PROGRAM PRG_Diagnostic
VAR
	i: UDINT;
	StAlr	 : ARRAY[0..CNC.NUM_STATIONS+4] OF ARRAY[0..CNC.NUM_MAX_STATION_ALARMS-1] OF BOOL;
	fbEVSt00 : ARRAY[0..CNC.NUM_MAX_MANUALS_00-1] OF FB_PneumaticActuator_2EV_Diagnostic;
	fbEVSt01 : ARRAY[0..CNC.NUM_MAX_MANUALS_01-1] OF FB_PneumaticActuator_2EV_Diagnostic;
	fbEVSt02 : ARRAY[0..CNC.NUM_MAX_MANUALS_02-1] OF FB_PneumaticActuator_2EV_Diagnostic;
	fbEVSt03 : ARRAY[0..CNC.NUM_MAX_MANUALS_03-1] OF FB_PneumaticActuator_2EV_Diagnostic;
	fbEVSt04 : ARRAY[0..CNC.NUM_MAX_MANUALS_04-1] OF FB_PneumaticActuator_2EV_Diagnostic;
	fbEVSt05 : ARRAY[0..CNC.NUM_MAX_MANUALS_05-1] OF FB_PneumaticActuator_2EV_Diagnostic;
	fbEVSt06 : ARRAY[0..CNC.NUM_MAX_MANUALS_06-1] OF FB_PneumaticActuator_2EV_Diagnostic;
	fbEVSt07 : ARRAY[0..CNC.NUM_MAX_MANUALS_07-1] OF FB_PneumaticActuator_2EV_Diagnostic;
	fbEVSt08 : ARRAY[0..CNC.NUM_MAX_MANUALS_08-1] OF FB_PneumaticActuator_2EV_Diagnostic;
	fbEVSt09 : ARRAY[0..CNC.NUM_MAX_MANUALS_09-1] OF FB_PneumaticActuator_2EV_Diagnostic;
	fbEVSt10 : ARRAY[0..CNC.NUM_MAX_MANUALS_10-1] OF FB_PneumaticActuator_2EV_Diagnostic;
	fbEVSt11 : ARRAY[0..CNC.NUM_MAX_MANUALS_11-1] OF FB_PneumaticActuator_2EV_Diagnostic;
	fbEVSt12 : ARRAY[0..CNC.NUM_MAX_MANUALS_12-1] OF FB_PneumaticActuator_2EV_Diagnostic;
	fbEVSt13 : ARRAY[0..CNC.NUM_MAX_MANUALS_13-1] OF FB_PneumaticActuator_2EV_Diagnostic;	
END_VAR

A_01_EVDiagnostic();
A_02_EVDiagnostic();
A_03_EVDiagnostic();
A_04_EVDiagnostic();
A_05_EVDiagnostic();
A_06_EVDiagnostic();
A_07_EVDiagnostic();
A_08_EVDiagnostic();
A_09_EVDiagnostic();
A_10_EVDiagnostic();
A_11_EVDiagnostic();
A_12_EVDiagnostic();
A_13_EVDiagnostic();

A_01_Alarms();

ACTION A_00_Alarms:
FOR i:= 0 TO CNC.NUM_MAX_STATION_ALARMS -1 DO 
	StAlr[0][i] := PRG_EventManagement._PMCEventCollectors._CheckFanucPMCActiveAlarmList_St00_Alr._PMCEvents[i].bRaised;
END_FOR

HMI.St0.EVInfo[64].Error := PRG_Diagnostic.fbEVSt00[0].Q_eStatus = eEV_Status.MovingForward AND StAlr[1][0];		
HMI.St0.EVInfo[65].Error := PRG_Diagnostic.fbEVSt00[0].Q_eStatus = eEV_Status.MovingBackward AND StAlr[1][0];
HMI.St0.EVInfo[64].Error := PRG_Diagnostic.fbEVSt00[1].Q_eStatus = eEV_Status.MovingForward AND StAlr[1][0];
HMI.St0.EVInfo[65].Error := PRG_Diagnostic.fbEVSt00[1].Q_eStatus = eEV_Status.MovingBackward AND StAlr[1][0]; 
      
HMI.St0.EVInfo[66].dTime := PRG_Diagnostic.fbEVSt00[0].Q_tElapsedTimeFwd;		
HMI.St0.EVInfo[67].dTime := PRG_Diagnostic.fbEVSt00[0].Q_tElapsedTimeBwd;
HMI.St0.EVInfo[66].dTime := PRG_Diagnostic.fbEVSt00[1].Q_tElapsedTimeFwd;
HMI.St0.EVInfo[67].dTime := PRG_Diagnostic.fbEVSt00[1].Q_tElapsedTimeBwd;
END_ACTION

ACTION A_00_EVDiagnostic:
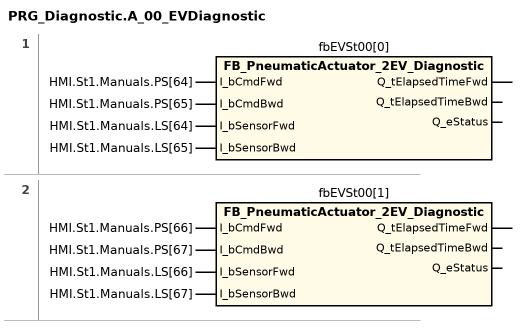
// NETWORK 1
fbEVSt00[0](
    I_bCmdFwd := HMI.St1.Manuals.PS[64],
    I_bCmdBwd := HMI.St1.Manuals.PS[65],
    I_bSensorFwd := HMI.St1.Manuals.LS[64],
    I_bSensorBwd := HMI.St1.Manuals.LS[65]); // FB_PneumaticActuator_2EV_Diagnostic

// NETWORK 2
fbEVSt00[1](
    I_bCmdFwd := HMI.St1.Manuals.PS[66],
    I_bCmdBwd := HMI.St1.Manuals.PS[67],
    I_bSensorFwd := HMI.St1.Manuals.LS[66],
    I_bSensorBwd := HMI.St1.Manuals.LS[67]); // FB_PneumaticActuator_2EV_Diagnostic
END_ACTION

ACTION A_01_Alarms:
FOR i:= 0 TO CNC.NUM_MAX_STATION_ALARMS -1 DO 
	StAlr[1][i] := PRG_EventManagement._PMCEventCollectors._CheckFanucPMCActiveAlarmList_St01_Alr._PMCEvents[i].bRaised;
END_FOR

HMI.St1.EVInfo[32].Error := PRG_Diagnostic.fbEVSt01[0].Q_eStatus = eEV_Status.MovingForward AND StAlr[1][0];		
HMI.St1.EVInfo[33].Error := PRG_Diagnostic.fbEVSt01[0].Q_eStatus = eEV_Status.MovingBackward AND StAlr[1][0];
HMI.St1.EVInfo[34].Error := PRG_Diagnostic.fbEVSt01[1].Q_eStatus = eEV_Status.MovingForward AND StAlr[1][0];
HMI.St1.EVInfo[35].Error := PRG_Diagnostic.fbEVSt01[1].Q_eStatus = eEV_Status.MovingBackward AND StAlr[1][0]; 
HMI.St1.EVInfo[36].Error := PRG_Diagnostic.fbEVSt01[2].Q_eStatus = eEV_Status.MovingForward AND StAlr[1][0];		
HMI.St1.EVInfo[37].Error := PRG_Diagnostic.fbEVSt01[2].Q_eStatus = eEV_Status.MovingBackward AND StAlr[1][0]; 
HMI.St1.EVInfo[25].Error := PRG_Diagnostic.fbEVSt01[3].Q_eStatus = eEV_Status.MovingForward AND StAlr[1][0];		
HMI.St1.EVInfo[26].Error := PRG_Diagnostic.fbEVSt01[3].Q_eStatus = eEV_Status.MovingBackward AND StAlr[1][0]; 

HMI.St1.EVInfo[32].dTime := PRG_Diagnostic.fbEVSt01[0].Q_tElapsedTimeFwd;		
HMI.St1.EVInfo[33].dTime := PRG_Diagnostic.fbEVSt01[0].Q_tElapsedTimeBwd;
HMI.St1.EVInfo[34].dTime := PRG_Diagnostic.fbEVSt01[1].Q_tElapsedTimeFwd;
HMI.St1.EVInfo[35].dTime := PRG_Diagnostic.fbEVSt01[1].Q_tElapsedTimeBwd;
HMI.St1.EVInfo[36].dTime := PRG_Diagnostic.fbEVSt01[2].Q_tElapsedTimeFwd;		
HMI.St1.EVInfo[37].dTime := PRG_Diagnostic.fbEVSt01[2].Q_tElapsedTimeBwd;
HMI.St1.EVInfo[25].dTime := PRG_Diagnostic.fbEVSt01[3].Q_tElapsedTimeFwd;		
HMI.St1.EVInfo[26].dTime := PRG_Diagnostic.fbEVSt01[3].Q_tElapsedTimeBwd;
END_ACTION

ACTION A_01_EVDiagnostic:
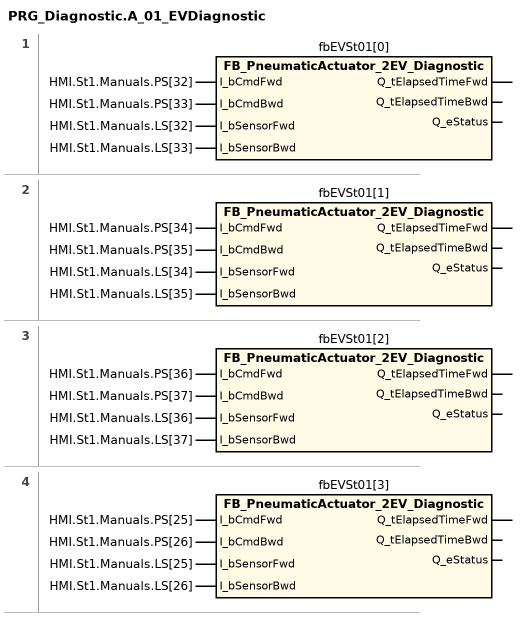
// NETWORK 1
fbEVSt01[0](
    I_bCmdFwd := HMI.St1.Manuals.PS[32],
    I_bCmdBwd := HMI.St1.Manuals.PS[33],
    I_bSensorFwd := HMI.St1.Manuals.LS[32],
    I_bSensorBwd := HMI.St1.Manuals.LS[33]); // FB_PneumaticActuator_2EV_Diagnostic

// NETWORK 2
fbEVSt01[1](
    I_bCmdFwd := HMI.St1.Manuals.PS[34],
    I_bCmdBwd := HMI.St1.Manuals.PS[35],
    I_bSensorFwd := HMI.St1.Manuals.LS[34],
    I_bSensorBwd := HMI.St1.Manuals.LS[35]); // FB_PneumaticActuator_2EV_Diagnostic

// NETWORK 3
fbEVSt01[2](
    I_bCmdFwd := HMI.St1.Manuals.PS[36],
    I_bCmdBwd := HMI.St1.Manuals.PS[37],
    I_bSensorFwd := HMI.St1.Manuals.LS[36],
    I_bSensorBwd := HMI.St1.Manuals.LS[37]); // FB_PneumaticActuator_2EV_Diagnostic

// NETWORK 4
fbEVSt01[3](
    I_bCmdFwd := HMI.St1.Manuals.PS[25],
    I_bCmdBwd := HMI.St1.Manuals.PS[26],
    I_bSensorFwd := HMI.St1.Manuals.LS[25],
    I_bSensorBwd := HMI.St1.Manuals.LS[26]); // FB_PneumaticActuator_2EV_Diagnostic
END_ACTION

ACTION A_02_Alarms:
FOR i:= 0 TO CNC.NUM_MAX_STATION_ALARMS -1 DO 
	StAlr[2][i] := PRG_EventManagement._PMCEventCollectors._CheckFanucPMCActiveAlarmList_St02_Alr._PMCEvents[i].bRaised;
END_FOR

HMI.St2.EVInfo[32].Error := PRG_Diagnostic.fbEVSt02[0].Q_eStatus = eEV_Status.MovingForward  AND StAlr[2][0];		
HMI.St2.EVInfo[33].Error := PRG_Diagnostic.fbEVSt02[0].Q_eStatus = eEV_Status.MovingBackward AND StAlr[2][0];
HMI.St2.EVInfo[34].Error := PRG_Diagnostic.fbEVSt02[1].Q_eStatus = eEV_Status.MovingForward  AND StAlr[2][0];
HMI.St2.EVInfo[35].Error := PRG_Diagnostic.fbEVSt02[1].Q_eStatus = eEV_Status.MovingBackward AND StAlr[2][0]; 
                                                  
HMI.St2.EVInfo[32].dTime := PRG_Diagnostic.fbEVSt02[0].Q_tElapsedTimeFwd;		
HMI.St2.EVInfo[33].dTime := PRG_Diagnostic.fbEVSt02[0].Q_tElapsedTimeBwd;
HMI.St2.EVInfo[34].dTime := PRG_Diagnostic.fbEVSt02[1].Q_tElapsedTimeFwd;
HMI.St2.EVInfo[35].dTime := PRG_Diagnostic.fbEVSt02[1].Q_tElapsedTimeBwd;
END_ACTION

ACTION A_02_EVDiagnostic:
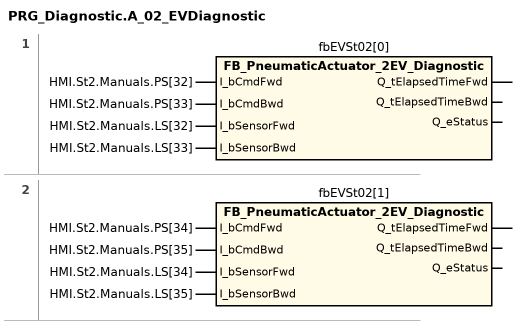
// NETWORK 1
fbEVSt02[0](
    I_bCmdFwd := HMI.St2.Manuals.PS[32],
    I_bCmdBwd := HMI.St2.Manuals.PS[33],
    I_bSensorFwd := HMI.St2.Manuals.LS[32],
    I_bSensorBwd := HMI.St2.Manuals.LS[33]); // FB_PneumaticActuator_2EV_Diagnostic

// NETWORK 2
fbEVSt02[1](
    I_bCmdFwd := HMI.St2.Manuals.PS[34],
    I_bCmdBwd := HMI.St2.Manuals.PS[35],
    I_bSensorFwd := HMI.St2.Manuals.LS[34],
    I_bSensorBwd := HMI.St2.Manuals.LS[35]); // FB_PneumaticActuator_2EV_Diagnostic
END_ACTION

ACTION A_03_Alarms:
FOR i:= 0 TO CNC.NUM_MAX_STATION_ALARMS -1 DO 
	StAlr[3][i] := PRG_EventManagement._PMCEventCollectors._CheckFanucPMCActiveAlarmList_St03_Alr._PMCEvents[i].bRaised;
END_FOR

HMI.St3.EVInfo[33].Error := PRG_Diagnostic.fbEVSt03[0].Q_eStatus = eEV_Status.MovingForward  AND StAlr[3][0];		
HMI.St3.EVInfo[32].Error := PRG_Diagnostic.fbEVSt03[0].Q_eStatus = eEV_Status.MovingBackward AND StAlr[3][0];
      
HMI.St3.EVInfo[33].dTime := PRG_Diagnostic.fbEVSt03[0].Q_tElapsedTimeFwd;		
HMI.St3.EVInfo[32].dTime := PRG_Diagnostic.fbEVSt03[0].Q_tElapsedTimeBwd;
END_ACTION

ACTION A_03_EVDiagnostic:
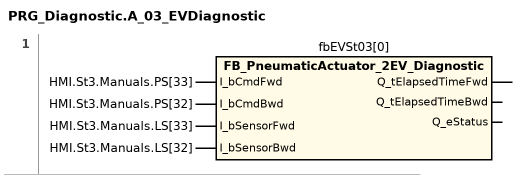
// NETWORK 1
fbEVSt03[0](
    I_bCmdFwd := HMI.St3.Manuals.PS[33],
    I_bCmdBwd := HMI.St3.Manuals.PS[32],
    I_bSensorFwd := HMI.St3.Manuals.LS[33],
    I_bSensorBwd := HMI.St3.Manuals.LS[32]); // FB_PneumaticActuator_2EV_Diagnostic
END_ACTION

ACTION A_04_Alarms:
FOR i:= 0 TO CNC.NUM_MAX_STATION_ALARMS -1 DO 
	StAlr[4][i] := PRG_EventManagement._PMCEventCollectors._CheckFanucPMCActiveAlarmList_St04_Alr._PMCEvents[i].bRaised;
END_FOR

HMI.St4.EVInfo[36].Error := PRG_Diagnostic.fbEVSt04[2].Q_eStatus = eEV_Status.MovingForward  AND StAlr[4][0];
HMI.St4.EVInfo[37].Error := PRG_Diagnostic.fbEVSt04[2].Q_eStatus = eEV_Status.MovingBackward AND StAlr[4][0]; 
HMI.St4.EVInfo[38].Error := PRG_Diagnostic.fbEVSt04[3].Q_eStatus = eEV_Status.MovingForward  AND StAlr[4][0];		
HMI.St4.EVInfo[39].Error := PRG_Diagnostic.fbEVSt04[3].Q_eStatus = eEV_Status.MovingBackward AND StAlr[4][0]; 
                                                  
HMI.St4.EVInfo[36].dTime := PRG_Diagnostic.fbEVSt04[2].Q_tElapsedTimeFwd;		
HMI.St4.EVInfo[37].dTime := PRG_Diagnostic.fbEVSt04[2].Q_tElapsedTimeBwd;
HMI.St4.EVInfo[38].dTime := PRG_Diagnostic.fbEVSt04[3].Q_tElapsedTimeFwd;
HMI.St4.EVInfo[39].dTime := PRG_Diagnostic.fbEVSt04[3].Q_tElapsedTimeBwd;
END_ACTION

ACTION A_04_EVDiagnostic:
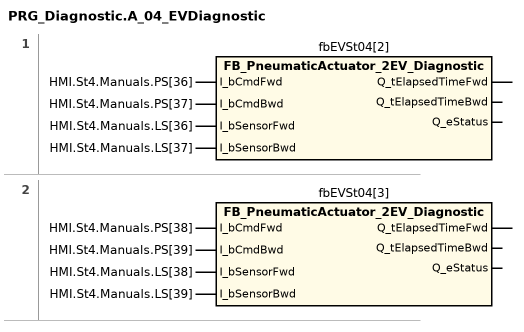
// NETWORK 1
fbEVSt04[2](
    I_bCmdFwd := HMI.St4.Manuals.PS[36],
    I_bCmdBwd := HMI.St4.Manuals.PS[37],
    I_bSensorFwd := HMI.St4.Manuals.LS[36],
    I_bSensorBwd := HMI.St4.Manuals.LS[37]); // FB_PneumaticActuator_2EV_Diagnostic

// NETWORK 2
fbEVSt04[3](
    I_bCmdFwd := HMI.St4.Manuals.PS[38],
    I_bCmdBwd := HMI.St4.Manuals.PS[39],
    I_bSensorFwd := HMI.St4.Manuals.LS[38],
    I_bSensorBwd := HMI.St4.Manuals.LS[39]); // FB_PneumaticActuator_2EV_Diagnostic
END_ACTION

ACTION A_05_Alarms:
FOR i:= 0 TO CNC.NUM_MAX_STATION_ALARMS -1 DO 
	StAlr[5][i] := PRG_EventManagement._PMCEventCollectors._CheckFanucPMCActiveAlarmList_St05_Alr._PMCEvents[i].bRaised;
END_FOR

HMI.St5.EVInfo[40].Error := PRG_Diagnostic.fbEVSt05[4].Q_eStatus  = eEV_Status.MovingForward  AND StAlr[5][0];		
HMI.St5.EVInfo[41].Error := PRG_Diagnostic.fbEVSt05[4].Q_eStatus  = eEV_Status.MovingBackward AND StAlr[5][0];
HMI.St5.EVInfo[64].Error := PRG_Diagnostic.fbEVSt05[16].Q_eStatus = eEV_Status.MovingForward  AND StAlr[5][0];
HMI.St5.EVInfo[65].Error := PRG_Diagnostic.fbEVSt05[16].Q_eStatus = eEV_Status.MovingBackward AND StAlr[5][0]; 
HMI.St5.EVInfo[66].Error := PRG_Diagnostic.fbEVSt05[17].Q_eStatus = eEV_Status.MovingForward  AND StAlr[5][0];		
HMI.St5.EVInfo[67].Error := PRG_Diagnostic.fbEVSt05[17].Q_eStatus = eEV_Status.MovingBackward AND StAlr[5][0]; 
                                                  
HMI.St5.EVInfo[40].dTime := PRG_Diagnostic.fbEVSt05[4].Q_tElapsedTimeFwd;		
HMI.St5.EVInfo[41].dTime := PRG_Diagnostic.fbEVSt05[4].Q_tElapsedTimeBwd;
HMI.St5.EVInfo[64].dTime := PRG_Diagnostic.fbEVSt05[16].Q_tElapsedTimeFwd;
HMI.St5.EVInfo[65].dTime := PRG_Diagnostic.fbEVSt05[16].Q_tElapsedTimeBwd;
HMI.St5.EVInfo[66].dTime := PRG_Diagnostic.fbEVSt05[17].Q_tElapsedTimeFwd;		
HMI.St5.EVInfo[67].dTime := PRG_Diagnostic.fbEVSt05[17].Q_tElapsedTimeBwd;
END_ACTION

ACTION A_05_EVDiagnostic:
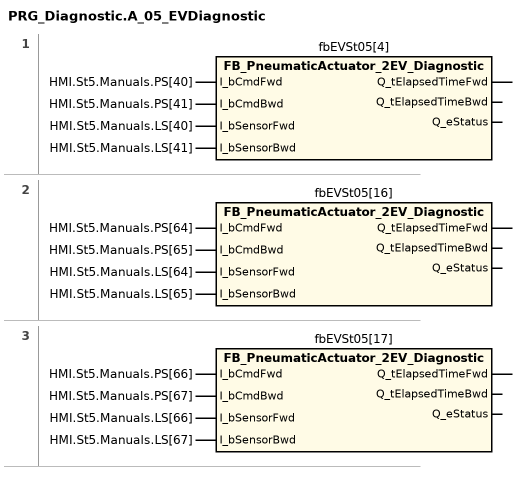
// NETWORK 1
fbEVSt05[4](
    I_bCmdFwd := HMI.St5.Manuals.PS[40],
    I_bCmdBwd := HMI.St5.Manuals.PS[41],
    I_bSensorFwd := HMI.St5.Manuals.LS[40],
    I_bSensorBwd := HMI.St5.Manuals.LS[41]); // FB_PneumaticActuator_2EV_Diagnostic

// NETWORK 2
fbEVSt05[16](
    I_bCmdFwd := HMI.St5.Manuals.PS[64],
    I_bCmdBwd := HMI.St5.Manuals.PS[65],
    I_bSensorFwd := HMI.St5.Manuals.LS[64],
    I_bSensorBwd := HMI.St5.Manuals.LS[65]); // FB_PneumaticActuator_2EV_Diagnostic

// NETWORK 3
fbEVSt05[17](
    I_bCmdFwd := HMI.St5.Manuals.PS[66],
    I_bCmdBwd := HMI.St5.Manuals.PS[67],
    I_bSensorFwd := HMI.St5.Manuals.LS[66],
    I_bSensorBwd := HMI.St5.Manuals.LS[67]); // FB_PneumaticActuator_2EV_Diagnostic
END_ACTION

ACTION A_06_Alarms:
FOR i:= 0 TO CNC.NUM_MAX_STATION_ALARMS -1 DO 
	StAlr[6][i] := PRG_EventManagement._PMCEventCollectors._CheckFanucPMCActiveAlarmList_St06_Alr._PMCEvents[i].bRaised;
END_FOR

HMI.St6.EVInfo[40].Error := PRG_Diagnostic.fbEVSt06[4].Q_eStatus = eEV_Status.MovingForward  AND StAlr[6][0];		
HMI.St6.EVInfo[41].Error := PRG_Diagnostic.fbEVSt06[4].Q_eStatus = eEV_Status.MovingBackward AND StAlr[6][0]; 

HMI.St6.EVInfo[40].dTime := PRG_Diagnostic.fbEVSt06[4].Q_tElapsedTimeFwd;		
HMI.St6.EVInfo[41].dTime := PRG_Diagnostic.fbEVSt06[4].Q_tElapsedTimeBwd;
END_ACTION

ACTION A_06_EVDiagnostic:
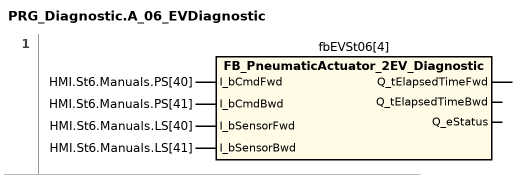
// NETWORK 1
fbEVSt06[4](
    I_bCmdFwd := HMI.St6.Manuals.PS[40],
    I_bCmdBwd := HMI.St6.Manuals.PS[41],
    I_bSensorFwd := HMI.St6.Manuals.LS[40],
    I_bSensorBwd := HMI.St6.Manuals.LS[41]); // FB_PneumaticActuator_2EV_Diagnostic
END_ACTION

ACTION A_07_Alarms:
FOR i:= 0 TO CNC.NUM_MAX_STATION_ALARMS -1 DO 
	StAlr[7][i] := PRG_EventManagement._PMCEventCollectors._CheckFanucPMCActiveAlarmList_St07_Alr._PMCEvents[i].bRaised;
END_FOR

HMI.St1.EVInfo[40].Error := PRG_Diagnostic.fbEVSt07[4].Q_eStatus = eEV_Status.MovingForward  AND StAlr[7][0];		
HMI.St1.EVInfo[41].Error := PRG_Diagnostic.fbEVSt07[4].Q_eStatus = eEV_Status.MovingBackward AND StAlr[7][0];

HMI.St1.EVInfo[40].dTime := PRG_Diagnostic.fbEVSt07[4].Q_tElapsedTimeFwd;		
HMI.St1.EVInfo[41].dTime := PRG_Diagnostic.fbEVSt07[4].Q_tElapsedTimeBwd;
END_ACTION

ACTION A_07_EVDiagnostic:
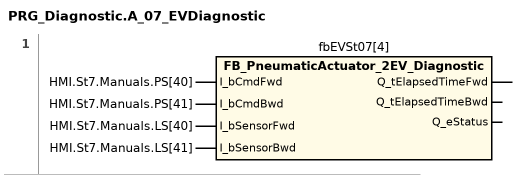
// NETWORK 1
fbEVSt07[4](
    I_bCmdFwd := HMI.St7.Manuals.PS[40],
    I_bCmdBwd := HMI.St7.Manuals.PS[41],
    I_bSensorFwd := HMI.St7.Manuals.LS[40],
    I_bSensorBwd := HMI.St7.Manuals.LS[41]); // FB_PneumaticActuator_2EV_Diagnostic
END_ACTION

ACTION A_08_Alarms:
FOR i:= 0 TO CNC.NUM_MAX_STATION_ALARMS -1 DO 
	StAlr[8][i] := PRG_EventManagement._PMCEventCollectors._CheckFanucPMCActiveAlarmList_St08_Alr._PMCEvents[i].bRaised;
END_FOR

HMI.St8.EVInfo[40].Error := PRG_Diagnostic.fbEVSt08[0].Q_eStatus = eEV_Status.MovingForward  AND StAlr[8][0];		
HMI.St8.EVInfo[41].Error := PRG_Diagnostic.fbEVSt08[0].Q_eStatus = eEV_Status.MovingBackward AND StAlr[8][0];

HMI.St8.EVInfo[40].dTime := PRG_Diagnostic.fbEVSt08[0].Q_tElapsedTimeFwd;		
HMI.St8.EVInfo[41].dTime := PRG_Diagnostic.fbEVSt08[0].Q_tElapsedTimeBwd;
END_ACTION

ACTION A_08_EVDiagnostic:
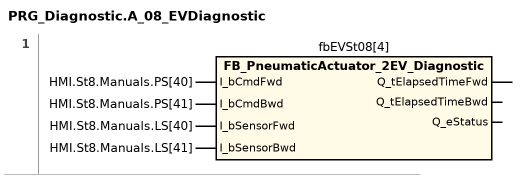
// NETWORK 1
fbEVSt08[4](
    I_bCmdFwd := HMI.St8.Manuals.PS[40],
    I_bCmdBwd := HMI.St8.Manuals.PS[41],
    I_bSensorFwd := HMI.St8.Manuals.LS[40],
    I_bSensorBwd := HMI.St8.Manuals.LS[41]); // FB_PneumaticActuator_2EV_Diagnostic
END_ACTION

ACTION A_09_Alarms:
FOR i:= 0 TO CNC.NUM_MAX_STATION_ALARMS -1 DO 
	StAlr[9][i] := PRG_EventManagement._PMCEventCollectors._CheckFanucPMCActiveAlarmList_St09_Alr._PMCEvents[i].bRaised;
END_FOR

HMI.St9.EVInfo[40].Error := PRG_Diagnostic.fbEVSt09[4].Q_eStatus = eEV_Status.MovingForward  AND StAlr[1][0];		
HMI.St9.EVInfo[41].Error := PRG_Diagnostic.fbEVSt09[4].Q_eStatus = eEV_Status.MovingBackward AND StAlr[1][0];

HMI.St9.EVInfo[40].dTime := PRG_Diagnostic.fbEVSt09[4].Q_tElapsedTimeFwd;		
HMI.St9.EVInfo[41].dTime := PRG_Diagnostic.fbEVSt09[4].Q_tElapsedTimeBwd;
END_ACTION

ACTION A_09_EVDiagnostic:
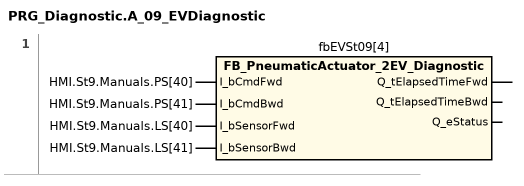
// NETWORK 1
fbEVSt09[4](
    I_bCmdFwd := HMI.St9.Manuals.PS[40],
    I_bCmdBwd := HMI.St9.Manuals.PS[41],
    I_bSensorFwd := HMI.St9.Manuals.LS[40],
    I_bSensorBwd := HMI.St9.Manuals.LS[41]); // FB_PneumaticActuator_2EV_Diagnostic
END_ACTION

ACTION A_10_Alarms:
FOR i:= 0 TO CNC.NUM_MAX_STATION_ALARMS -1 DO 
	StAlr[10][i] := PRG_EventManagement._PMCEventCollectors._CheckFanucPMCActiveAlarmList_St10_Alr._PMCEvents[i].bRaised;
END_FOR

HMI.St10.EVInfo[40].Error := PRG_Diagnostic.fbEVSt10[4].Q_eStatus = eEV_Status.MovingForward   AND StAlr[10][0];		
HMI.St10.EVInfo[41].Error := PRG_Diagnostic.fbEVSt10[4].Q_eStatus = eEV_Status.MovingBackward  AND StAlr[10][0];
HMI.St10.EVInfo[40].Error := PRG_Diagnostic.fbEVSt10[11].Q_eStatus = eEV_Status.MovingForward  AND StAlr[10][0];
HMI.St10.EVInfo[41].Error := PRG_Diagnostic.fbEVSt10[11].Q_eStatus = eEV_Status.MovingBackward AND StAlr[10][0]; 
                                                  
HMI.St10.EVInfo[54].dTime := PRG_Diagnostic.fbEVSt10[4].Q_tElapsedTimeFwd;		
HMI.St10.EVInfo[55].dTime := PRG_Diagnostic.fbEVSt10[4].Q_tElapsedTimeBwd;
HMI.St10.EVInfo[54].dTime := PRG_Diagnostic.fbEVSt10[11].Q_tElapsedTimeFwd;
HMI.St10.EVInfo[55].dTime := PRG_Diagnostic.fbEVSt10[11].Q_tElapsedTimeBwd;
END_ACTION

ACTION A_10_EVDiagnostic:
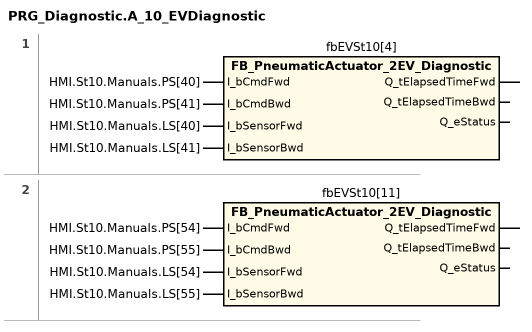
// NETWORK 1
fbEVSt10[4](
    I_bCmdFwd := HMI.St10.Manuals.PS[40],
    I_bCmdBwd := HMI.St10.Manuals.PS[41],
    I_bSensorFwd := HMI.St10.Manuals.LS[40],
    I_bSensorBwd := HMI.St10.Manuals.LS[41]); // FB_PneumaticActuator_2EV_Diagnostic

// NETWORK 2
fbEVSt10[11](
    I_bCmdFwd := HMI.St10.Manuals.PS[54],
    I_bCmdBwd := HMI.St10.Manuals.PS[55],
    I_bSensorFwd := HMI.St10.Manuals.LS[54],
    I_bSensorBwd := HMI.St10.Manuals.LS[55]); // FB_PneumaticActuator_2EV_Diagnostic
END_ACTION

ACTION A_11_Alarms:
FOR i:= 0 TO CNC.NUM_MAX_STATION_ALARMS -1 DO 
	StAlr[11][i] := PRG_EventManagement._PMCEventCollectors._CheckFanucPMCActiveAlarmList_St11_Alr._PMCEvents[i].bRaised;
END_FOR

HMI.St11.EVInfo[32].Error := PRG_Diagnostic.fbEVSt01[0].Q_eStatus = eEV_Status.MovingForward  AND StAlr[11][0];		
HMI.St11.EVInfo[33].Error := PRG_Diagnostic.fbEVSt01[0].Q_eStatus = eEV_Status.MovingBackward AND StAlr[11][0];
HMI.St11.EVInfo[34].Error := PRG_Diagnostic.fbEVSt01[1].Q_eStatus = eEV_Status.MovingForward  AND StAlr[11][0];
HMI.St11.EVInfo[35].Error := PRG_Diagnostic.fbEVSt01[1].Q_eStatus = eEV_Status.MovingBackward AND StAlr[11][0]; 

HMI.St11.EVInfo[32].dTime := PRG_Diagnostic.fbEVSt01[0].Q_tElapsedTimeFwd;		
HMI.St11.EVInfo[33].dTime := PRG_Diagnostic.fbEVSt01[0].Q_tElapsedTimeBwd;
HMI.St11.EVInfo[34].dTime := PRG_Diagnostic.fbEVSt01[1].Q_tElapsedTimeFwd;
HMI.St11.EVInfo[35].dTime := PRG_Diagnostic.fbEVSt01[1].Q_tElapsedTimeBwd;
END_ACTION

ACTION A_11_EVDiagnostic:
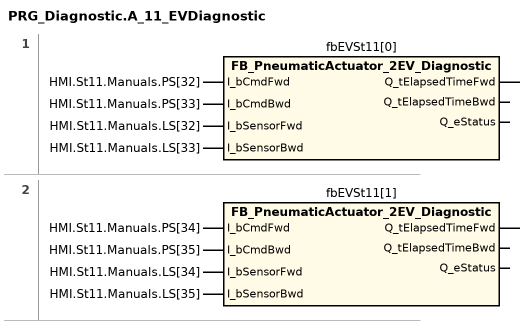
// NETWORK 1
fbEVSt11[0](
    I_bCmdFwd := HMI.St11.Manuals.PS[32],
    I_bCmdBwd := HMI.St11.Manuals.PS[33],
    I_bSensorFwd := HMI.St11.Manuals.LS[32],
    I_bSensorBwd := HMI.St11.Manuals.LS[33]); // FB_PneumaticActuator_2EV_Diagnostic

// NETWORK 2
fbEVSt11[1](
    I_bCmdFwd := HMI.St11.Manuals.PS[34],
    I_bCmdBwd := HMI.St11.Manuals.PS[35],
    I_bSensorFwd := HMI.St11.Manuals.LS[34],
    I_bSensorBwd := HMI.St11.Manuals.LS[35]); // FB_PneumaticActuator_2EV_Diagnostic
END_ACTION

ACTION A_12_Alarms:
FOR i:= 0 TO CNC.NUM_MAX_STATION_ALARMS -1 DO 
	StAlr[12][i] := PRG_EventManagement._PMCEventCollectors._CheckFanucPMCActiveAlarmList_St12_Alr._PMCEvents[i].bRaised;
END_FOR

HMI.St12.EVInfo[32].Error := PRG_Diagnostic.fbEVSt12[0].Q_eStatus = eEV_Status.MovingForward  AND StAlr[12][0];		
HMI.St12.EVInfo[33].Error := PRG_Diagnostic.fbEVSt12[0].Q_eStatus = eEV_Status.MovingBackward AND StAlr[12][0];
HMI.St12.EVInfo[34].Error := PRG_Diagnostic.fbEVSt12[1].Q_eStatus = eEV_Status.MovingForward  AND StAlr[12][0];
HMI.St12.EVInfo[35].Error := PRG_Diagnostic.fbEVSt12[1].Q_eStatus = eEV_Status.MovingBackward AND StAlr[12][0]; 
HMI.St12.EVInfo[36].Error := PRG_Diagnostic.fbEVSt12[2].Q_eStatus = eEV_Status.MovingForward  AND StAlr[12][0];		
HMI.St12.EVInfo[37].Error := PRG_Diagnostic.fbEVSt12[2].Q_eStatus = eEV_Status.MovingBackward AND StAlr[12][0];
HMI.St12.EVInfo[38].Error := PRG_Diagnostic.fbEVSt12[3].Q_eStatus = eEV_Status.MovingForward  AND StAlr[12][0];		
HMI.St12.EVInfo[39].Error := PRG_Diagnostic.fbEVSt12[3].Q_eStatus = eEV_Status.MovingBackward AND StAlr[12][0];
HMI.St12.EVInfo[40].Error := PRG_Diagnostic.fbEVSt12[4].Q_eStatus = eEV_Status.MovingForward  AND StAlr[12][0];		
HMI.St12.EVInfo[41].Error := PRG_Diagnostic.fbEVSt12[4].Q_eStatus = eEV_Status.MovingBackward AND StAlr[12][0]; 

HMI.St12.EVInfo[32].dTime := PRG_Diagnostic.fbEVSt12[0].Q_tElapsedTimeFwd;		
HMI.St12.EVInfo[33].dTime := PRG_Diagnostic.fbEVSt12[0].Q_tElapsedTimeBwd;
HMI.St12.EVInfo[34].dTime := PRG_Diagnostic.fbEVSt12[1].Q_tElapsedTimeFwd;
HMI.St12.EVInfo[35].dTime := PRG_Diagnostic.fbEVSt12[1].Q_tElapsedTimeBwd;
HMI.St12.EVInfo[36].dTime := PRG_Diagnostic.fbEVSt12[2].Q_tElapsedTimeFwd;		
HMI.St12.EVInfo[37].dTime := PRG_Diagnostic.fbEVSt12[2].Q_tElapsedTimeBwd;
HMI.St12.EVInfo[38].dTime := PRG_Diagnostic.fbEVSt12[3].Q_tElapsedTimeFwd;		
HMI.St12.EVInfo[39].dTime := PRG_Diagnostic.fbEVSt12[3].Q_tElapsedTimeBwd;
HMI.St12.EVInfo[40].dTime := PRG_Diagnostic.fbEVSt12[4].Q_tElapsedTimeFwd;		
HMI.St12.EVInfo[41].dTime := PRG_Diagnostic.fbEVSt12[4].Q_tElapsedTimeBwd;
END_ACTION

ACTION A_12_EVDiagnostic:
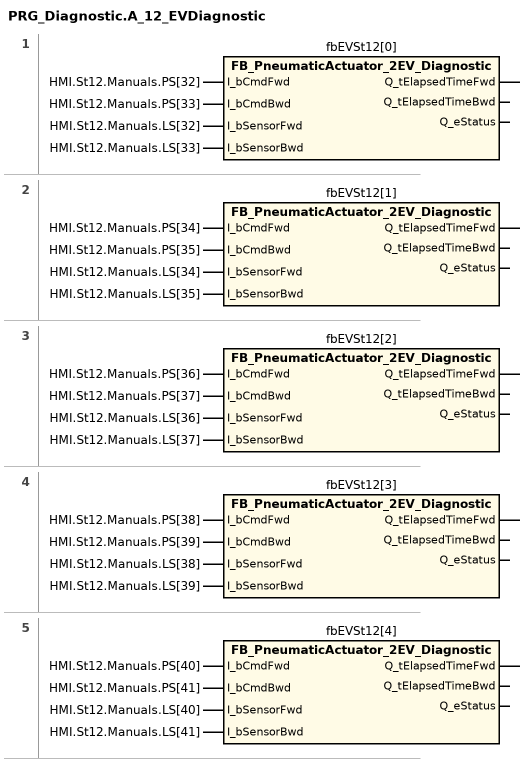
// NETWORK 1
fbEVSt12[0](
    I_bCmdFwd := HMI.St12.Manuals.PS[32],
    I_bCmdBwd := HMI.St12.Manuals.PS[33],
    I_bSensorFwd := HMI.St12.Manuals.LS[32],
    I_bSensorBwd := HMI.St12.Manuals.LS[33]); // FB_PneumaticActuator_2EV_Diagnostic

// NETWORK 2
fbEVSt12[1](
    I_bCmdFwd := HMI.St12.Manuals.PS[34],
    I_bCmdBwd := HMI.St12.Manuals.PS[35],
    I_bSensorFwd := HMI.St12.Manuals.LS[34],
    I_bSensorBwd := HMI.St12.Manuals.LS[35]); // FB_PneumaticActuator_2EV_Diagnostic

// NETWORK 3
fbEVSt12[2](
    I_bCmdFwd := HMI.St12.Manuals.PS[36],
    I_bCmdBwd := HMI.St12.Manuals.PS[37],
    I_bSensorFwd := HMI.St12.Manuals.LS[36],
    I_bSensorBwd := HMI.St12.Manuals.LS[37]); // FB_PneumaticActuator_2EV_Diagnostic

// NETWORK 4
fbEVSt12[3](
    I_bCmdFwd := HMI.St12.Manuals.PS[38],
    I_bCmdBwd := HMI.St12.Manuals.PS[39],
    I_bSensorFwd := HMI.St12.Manuals.LS[38],
    I_bSensorBwd := HMI.St12.Manuals.LS[39]); // FB_PneumaticActuator_2EV_Diagnostic

// NETWORK 5
fbEVSt12[4](
    I_bCmdFwd := HMI.St12.Manuals.PS[40],
    I_bCmdBwd := HMI.St12.Manuals.PS[41],
    I_bSensorFwd := HMI.St12.Manuals.LS[40],
    I_bSensorBwd := HMI.St12.Manuals.LS[41]); // FB_PneumaticActuator_2EV_Diagnostic
END_ACTION

ACTION A_13_Alarms:
FOR i:= 0 TO CNC.NUM_MAX_STATION_ALARMS -1 DO 
	StAlr[13][i] := PRG_EventManagement._PMCEventCollectors._CheckFanucPMCActiveAlarmList_St13_Alr._PMCEvents[i].bRaised;
END_FOR

HMI.St13.EVInfo[32].Error := PRG_Diagnostic.fbEVSt13[0].Q_eStatus = eEV_Status.MovingForward  AND StAlr[13][0];		
HMI.St13.EVInfo[33].Error := PRG_Diagnostic.fbEVSt13[0].Q_eStatus = eEV_Status.MovingBackward AND StAlr[13][0];
HMI.St13.EVInfo[34].Error := PRG_Diagnostic.fbEVSt13[1].Q_eStatus = eEV_Status.MovingForward  AND StAlr[13][0];
HMI.St13.EVInfo[35].Error := PRG_Diagnostic.fbEVSt13[1].Q_eStatus = eEV_Status.MovingBackward AND StAlr[13][0]; 
HMI.St13.EVInfo[36].Error := PRG_Diagnostic.fbEVSt13[2].Q_eStatus = eEV_Status.MovingForward  AND StAlr[13][0];		
HMI.St13.EVInfo[37].Error := PRG_Diagnostic.fbEVSt13[2].Q_eStatus = eEV_Status.MovingBackward AND StAlr[13][0]; 
HMI.St13.EVInfo[38].Error := PRG_Diagnostic.fbEVSt13[3].Q_eStatus = eEV_Status.MovingForward  AND StAlr[13][0];		
HMI.St13.EVInfo[39].Error := PRG_Diagnostic.fbEVSt13[3].Q_eStatus = eEV_Status.MovingBackward AND StAlr[13][0]; 

HMI.St13.EVInfo[32].dTime := PRG_Diagnostic.fbEVSt13[0].Q_tElapsedTimeFwd;		
HMI.St13.EVInfo[33].dTime := PRG_Diagnostic.fbEVSt13[0].Q_tElapsedTimeBwd;
HMI.St13.EVInfo[34].dTime := PRG_Diagnostic.fbEVSt13[1].Q_tElapsedTimeFwd;
HMI.St13.EVInfo[35].dTime := PRG_Diagnostic.fbEVSt13[1].Q_tElapsedTimeBwd;
HMI.St13.EVInfo[36].dTime := PRG_Diagnostic.fbEVSt13[2].Q_tElapsedTimeFwd;		
HMI.St13.EVInfo[37].dTime := PRG_Diagnostic.fbEVSt13[2].Q_tElapsedTimeBwd;
HMI.St13.EVInfo[38].dTime := PRG_Diagnostic.fbEVSt13[3].Q_tElapsedTimeFwd;		
HMI.St13.EVInfo[39].dTime := PRG_Diagnostic.fbEVSt13[3].Q_tElapsedTimeBwd;
END_ACTION

ACTION A_13_EVDiagnostic:
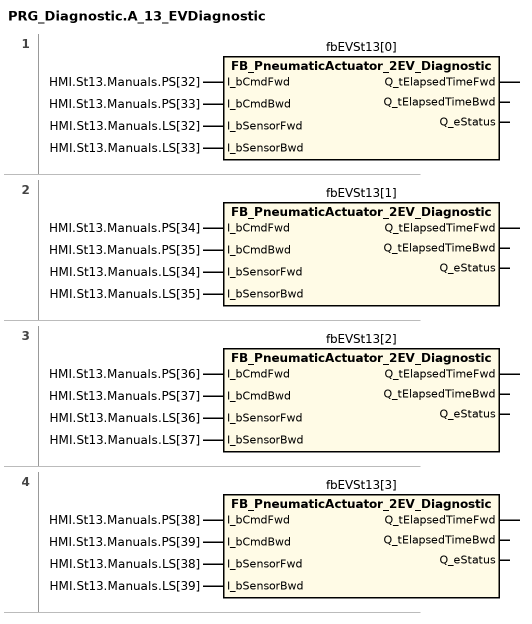
// NETWORK 1
fbEVSt13[0](
    I_bCmdFwd := HMI.St13.Manuals.PS[32],
    I_bCmdBwd := HMI.St13.Manuals.PS[33],
    I_bSensorFwd := HMI.St13.Manuals.LS[32],
    I_bSensorBwd := HMI.St13.Manuals.LS[33]); // FB_PneumaticActuator_2EV_Diagnostic

// NETWORK 2
fbEVSt13[1](
    I_bCmdFwd := HMI.St13.Manuals.PS[34],
    I_bCmdBwd := HMI.St13.Manuals.PS[35],
    I_bSensorFwd := HMI.St13.Manuals.LS[34],
    I_bSensorBwd := HMI.St13.Manuals.LS[35]); // FB_PneumaticActuator_2EV_Diagnostic

// NETWORK 3
fbEVSt13[2](
    I_bCmdFwd := HMI.St13.Manuals.PS[36],
    I_bCmdBwd := HMI.St13.Manuals.PS[37],
    I_bSensorFwd := HMI.St13.Manuals.LS[36],
    I_bSensorBwd := HMI.St13.Manuals.LS[37]); // FB_PneumaticActuator_2EV_Diagnostic

// NETWORK 4
fbEVSt13[3](
    I_bCmdFwd := HMI.St13.Manuals.PS[38],
    I_bCmdBwd := HMI.St13.Manuals.PS[39],
    I_bSensorFwd := HMI.St13.Manuals.LS[38],
    I_bSensorBwd := HMI.St13.Manuals.LS[39]); // FB_PneumaticActuator_2EV_Diagnostic
END_ACTION

END_PROGRAM

(* stored: Version 1.1.0.1, ProductVersion 3.1.4024.15
   POU PRG_Diagnostic: Id {adc91861-aa55-4305-bfac-bd2b856a148e}, SpecialFunc None
   Action A_00_Alarms: Id {18c0b9bd-8ae9-4423-847e-db8238966453}
   Action A_00_EVDiagnostic: Id {59c9defa-d32a-4095-aa94-e7b90637144f}
   Action A_01_Alarms: Id {24727d9b-13c9-4222-9961-ff712a4c9358}
   Action A_01_EVDiagnostic: Id {88fcfb40-2b85-4632-a930-2deb89fcff3e}
   Action A_02_Alarms: Id {b0148c85-5ccf-4e62-bb15-5fd4490b1a3a}
   Action A_02_EVDiagnostic: Id {488b1e0b-e364-4a56-868e-4b715e806523}
   Action A_03_Alarms: Id {dc5e5318-976e-4aff-905f-e35ce54c1fa3}
   Action A_03_EVDiagnostic: Id {c65fc63d-e765-4de2-a2b2-de392bd02c41}
   Action A_04_Alarms: Id {2e649310-b2f7-46c7-9f7f-5f39d85c2cfe}
   Action A_04_EVDiagnostic: Id {33ff257b-e0be-41a1-b077-6788c6211c65}
   Action A_05_Alarms: Id {db30b7c5-0a66-4db8-99b7-49a24148fc39}
   Action A_05_EVDiagnostic: Id {633d0ae6-5d64-449f-80ab-1d40a5d241c1}
   Action A_06_Alarms: Id {08d61cf6-7dc6-41c2-b43c-42e98bad5e91}
   Action A_06_EVDiagnostic: Id {1d8e3aef-321e-4b57-b89b-80fbc3f00db1}
   Action A_07_Alarms: Id {7d24a20d-c7aa-4a14-8f7a-5520127ce249}
   Action A_07_EVDiagnostic: Id {ab2d572e-8695-4611-9be4-f5f424167858}
   Action A_08_Alarms: Id {d123c85d-1bda-4ea8-b188-9fa38e8616e3}
   Action A_08_EVDiagnostic: Id {e70d8c2a-065d-46a8-b81c-3c51c956eae3}
   Action A_09_Alarms: Id {3f4cd056-7113-4baa-ab49-ccb87f8beed9}
   Action A_09_EVDiagnostic: Id {21abfc5d-39da-469c-b741-defb92c259f2}
   Action A_10_Alarms: Id {f8939af0-0049-429f-94af-99d90b1513a9}
   Action A_10_EVDiagnostic: Id {5fd81eb6-538d-4ac1-aec1-62c8c2fb5f59}
   Action A_11_Alarms: Id {d6ee8ec4-1efb-4b7a-a73f-71b95ed6e2f4}
   Action A_11_EVDiagnostic: Id {8ba0fc5c-53dd-4fe3-a9ab-39a6545575aa}
   Action A_12_Alarms: Id {d8835ecc-4e73-44a8-a024-3b975b0d16f7}
   Action A_12_EVDiagnostic: Id {36310899-d7cc-4648-b33d-aae0ee8059bf}
   Action A_13_Alarms: Id {45777c04-d760-44b9-9f98-a58a56e0869d}
   Action A_13_EVDiagnostic: Id {842e298a-aed1-4e78-89c9-34f641ba9a0a} *)
